Staubli VAL3: COM.pgx

public program COM(num& x_value[])
// Each bit is complemented: 1s become 0s and 0s become 1s.
  local string sBin
  local num l_idx
  local string sCom
begin
  if bDebug
    putln("COM()")
  endIf
  call decToBin(x_value,sBin)
  sCom=""
  for l_idx=0 to (len(sBin)-1)
    if mid(sBin,1,l_idx)=="1"
      sCom=sCom+"0"
    else
      sCom=sCom+"1"
    endIf
  endFor
  call binToDec(sCom,x_value)
end
